// TIA Portal V21 export
TYPE "Std_stMotore"
   STRUCT
      In : Struct   // Ingressi
         FbDigitali : Struct   // Feedback digitali
            WarningInverter : Bool;
            SezMotoreAperto : Bool;   // Sezionatore motore aperto 1 = Allarme
            Sovracorrente : Bool;   // Sovracorrente Motore
            CoppiaSuperata : Bool;   // Copia Superata
            FaultInverter : Bool;   // Fault from inverter
            FeedbackMarcia : Bool;   // Feedback di marcia
            TermicoIntervenuto : Bool;   // Termico Intervenuto
            TermicoServoventilazione : Bool;   // Termico servoventola intervenuto
            PulsantieraLocale : Struct
               Auto : Bool;   // Da HMI Automatico Selezionato
               Stop : Bool;
               ManPos : Bool;   // Da HMI Manuale positivo
               ManNeg : Bool;   // Da HMI Manuale negativo
               StatoFromPuls : Int;
            END_STRUCT;
         END_STRUCT;
         Reset : Bool;   // Reset
         ProfinetHwSubModule : HW_SUBMODULE;   // Indirizzo Periferica Hardward
         CmdPosRich : Bool;   // Comando positivo richiesto
         CmdNegRich : Bool;   // Comando negativo richiesto
         CmdVelocitaRich : Real;   // Velocità Richiesta (Hz)
         CmdPosizioneRich : Real;   // Posizione richiesta espressa in mm*1000
         ConsMovimentoPos : Bool;   // Abilitazione del motore a girare in direzione positiva
         ConsMovimentoNeg : Bool;   // Abilitazione del motore a girare in direzione negativa
      END_STRUCT;
      Prm : Struct   // Parametri
         Generali : Struct
            TStart { S7_SetPoint := 'True'} : "Std_stTimer";   // Ritardo Marcia
            Tstop { S7_SetPoint := 'True'} : "Std_stTimer";   // Ritardo Arresto
            TimeOutMarcia { S7_SetPoint := 'True'} : "Std_stTimer";   // Ritardo Controllo Feedback Marcia
            TStopServoventola { S7_SetPoint := 'True'} : "Std_stTimer";
            MassimaFrequenza { S7_SetPoint := 'True'} : Real;   // Massima frequenza per motore
            MinimaFrequenza : Real;   // Minima frequenza per motore
            Accellerazione : Real;   // Rampa Accelerazione Richiesta 100 = 1s
            Decellerazione : Real;   // Rampa Deceleraione Richiesta 100 = 1s
            InversioneRotazione : Bool;   // Inversione del senso di marcia in uscita motore
            K_Analogica : Int;   // Feedback speed
            K_TipoMotore : Int;
            K_VistaManuale : Int;
            Inverter : Struct
               MinimaFreqDel_Inv : Real;   // Minima frequenza impostato nell'inverter
               MassimaFreqDel_Inv : Real;   // Massima frequenza impostato nell'inverter
               Presente : Bool;
            END_STRUCT;
            Feedbackspeed_Virtuale : Bool;
         END_STRUCT;
         Abilitazioni : Struct
            Servoventilazione : Bool;
         END_STRUCT;
         Posizionatore : Struct
            KConv_HzSpeed : Real;
            DeadBand_InPosition : Real;
            LimiteFisicoPos : Real;
            LimiteFisicoNeg : Real;
         END_STRUCT;
         Quote : Array[0.."K_NumCamma"] of Real;
         UnitàMisura : "Std_UnitàDiMisura";
      END_STRUCT;
      Hmi : Struct   // Selezioni HMI
         STW1 : Word;   // Mostra a schermo lo status word dell'inverter inverter
         CTW1 : Word;   // Mostra a schermo la control word dell'inverter inverter
         TipoManuale : Int;
         StatoCmd : Struct   // Da HMI
            StatoFromHmi : Byte;   // 0=Stop 1=Auto 2=ManPos 3=ManNeg
            Auto : Bool;   // Da HMI Automatico Selezionato
            Stop : Bool;
            ManPos : Bool;   // Da HMI Manuale positivo
            ManNeg : Bool;   // Da HMI Manuale negativo
            TestServoVentola : Bool;   // Test rotazione servoventilazione motore
         END_STRUCT;
         StatoMotore : Int;   // 0=StopAuto 1=Automatico 2=StopMan 3=Man 4=Allarme
         VelManuale : Real;
         Visibilita : Struct
            VelManuale : Bool;
            Posizioni : Bool;
            Servoventola : Bool;
         END_STRUCT;
         EseguiHomingAsse : Bool;
         CmdPosRich : Bool;
         CmdNegRich : Bool;
         BypassSicurezze : Bool;
      END_STRUCT;
      Dati : Struct
         Feedback_Speed : Real;
         Feedback_Marcia : Bool;   // Feedback di marcia
         WarningInverter : Bool;
         SensoMarciaPos : Bool;   // Marcia Avanti
         SensoMarciaNeg : Bool;   // Marcia Indietro
         Abilita : Bool;   // Abilitazione
         RetVal_Read_Inv : Int;
         RetVal_SCR_Inv : Int;
         PosRich_old : DInt;
         StatoMotoreOld : Int;
         PulsantieraLocalePresente : Bool;
         BloccoRichiamato : Bool;
         VelocitàDaInverter : DInt;
         FrequenzaRichiesta : Real;
         InclusoInUnaSequenza : Bool;
      END_STRUCT;
      Allarmi : Struct   // Allarmi Attivi
         "A" : Array[0.."K_NumAllarmiPerMotori"] of "Std_PrmAllarmeStd";
         WordHMI : Word;   // Word per lista segnalazioni HMI
      END_STRUCT;
      Out : Struct   // Uscite
         Pronto : Bool;   // Pronto Alla Marcia
         Allarme : Bool;   // Allarme Presente
         Avviso : Bool;   // Avviso Presente
         InMarcia : Bool;   // In Marcia
         CmdPosMotore : Bool;   // Comando positivo avanti salita
         CmdNegMotore : Bool;   // Comando negativo indeitro discesa
         CmdPosServoVentola : Bool;
         InMarciaRifRag : Bool;   // In Marcia Velocità Riferimento Raggiunta
         PosiRichiestaRaggiunta : Bool;
         Paw : Word;   // Velocita Attuale
         PosAttuale : Real;
         ErrCom : Int;   // Errore Comunicaiznoe
         CodiceAllarmeInv : DInt;   // Codice Allarme Sul Drive
         CodiceWarningInv : DInt;
         CorrenteAtt : Real;   // Corrente Attuale 0 - 10000
         InPosQuota : Array[0.."K_NumCamma"] of Bool;
      END_STRUCT;
      Rif_Inc : Struct   // Serve per sapere chi legge e scrive
         K_Pid : Int;
         K_Zona : Int := 0;
         K_Analogica : Int;   // Utilizzato per il feedback speed
         K_Sequenza : Array[0.."K_NumRifIncrociatiSequenza"] of Int;
      END_STRUCT;
   END_STRUCT;
   // // Allarmi."A"[1] : Comunicazione
   // // Allarmi."A"[2] : DriveInAllarme
   // // Allarmi."A"[3] : Sovracorrente
   // // Allarmi."A"[4] : Coppia
   // // Allarmi."A"[5] : Termico
   // // Allarmi."A"[6] : TimeOutMarcia
   // // Allarmi."A"[7] : SezMotoreAperto
   // // Allarmi."A"[8] : ScattoTermicoServoventola
   // // Allarmi."A"[9] : RichiestaAzzeramento
   // // Allarmi."A"[10] : LimiteFisicoPosRaggiunto
   // // Allarmi."A"[11] : LimiteFisicoNegRaggiunto
   // // Allarmi."A"[12] : MotoreNonInAutoDaHmi
   // // Allarmi."A"[13] : MotoreNonInAutoDaPulsLoc
END_TYPE
